TYPE Sensor :
STRUCT
	
END_STRUCT
END_TYPE

(* stored: Version 1.1.0.1, ProductVersion 3.1.4024.12
   DUT Sensor: Id {3fbdab91-883a-4964-a8c9-299b8d18c114} *)
